# B&R Automation Studio project Installer AS Technology Solution
Automation Studio 4.9

## Logical view

### Package Logical/Libraries - Global libraries

### Program Logical/Libraries/brdkSTR

#### brdkSTR_func.h
```c
#ifndef BRDK_STR_FUNCS
#define BRDK_STR_FUNCS 1

#include <brdkSTR.h>
#include <bur/plctypes.h>

#ifdef __cplusplus
	extern "C"
	{
#endif

#ifdef __cplusplus
	};
#endif

#endif
```

#### brdkStrAToUdint.c
```c
#include <brdkSTR_func.h>

unsigned long brdkStrAToUdint(unsigned long pString, unsigned char base) {
	unsigned long value = 0;
	signed long i, len = brdkStrLen(pString);
	if(len > 0) {
		for(i=0; i <len; i++) {
			switch(base) {

				case 0: case 10:
					if(((char*)pString)[i] >= 0x30 && ((char*)pString)[i] <= 0x39) value = (value * 10) + (((char*)pString)[i]-0x30);			/* 0x30 = 0, 0x39 = 9 */
					else {
						value = 0;
						i = len;
					}
					break;

				case 2:
					if(((char*)pString)[i] >= 0x30 && ((char*)pString)[i] <= 0x31) value += (((char*)pString)[i]-0x30)*(1<<(len-1-i));			/* 0x30 = 0, 0x31 = 1 */
					else {
						value = 0;
						i = len;
					}
					break;

				case 16:
					if(((char*)pString)[i] >= 0x30 && ((char*)pString)[i] <= 0x39) 	value += (((char*)pString)[i]-0x30)*(1<<(4*(len-1-i)));		/* 0x30 = 0, 0x39 = 9 */
					else if(((char*)pString)[i] >= 0x41 && ((char*)pString)[i] <= 0x46) value += (((char*)pString)[i]-0x37)*(1<<(4*(len-1-i)));	/* 0x41 = A, 0x46 = F */
					else if(((char*)pString)[i] >= 0x61 && ((char*)pString)[i] <= 0x66)value += (((char*)pString)[i]-0x57)*(1<<(4*(len-1-i)));	/* 0x61 = a, 0x66 = f */
					else {
						value = 0;
						i = len;
					}
					break;

				default:
					value = 0;
					i = len;
					break;

			}
		}
	}
	return value;
}
```

#### brdkStrSearch.c
```c
#include <brdkSTR_func.h>

signed long brdkStrSearch(unsigned long pString, unsigned long pSearchString) {
	signed long pos=-1, i=0,j=0, len1 = brdkStrLen(pString), len2 = brdkStrLen(pSearchString);

	if(len1>len2) {
		for(i=0; i <= len1-len2; i++) {
			j=0;
			if(((char*)pString)[i] == ((char*)pSearchString)[j]) {
				while(((char*)pString)[i+j] == ((char*)pSearchString)[j]) {
					j++;
					if(j==len2) {
						pos = i;
						i=len1-len2+1;
						break;
					}
				}
			}
		}
	}
	return pos;
}
```

### Library Logical/Libraries/TrkDiag (ANSIC)
Depends on: McAcpTrak

### Program Logical/Libraries/TrkPaper

#### TrkPaperShuttleControl.c
```c
#include <bur/plctypes.h>
#include <stdint.h>
#include <AsBrStr.h>

#define TRUE 1
#define FALSE 0

#ifdef __cplusplus
	extern "C"
	{
#endif
#include "TrkPaper.h"
#ifdef __cplusplus
	};
#endif

plcbit CheckValidity(char* selectedElem){
	char buf[2];
	//Get a substring of the first 3 characters
	brdkStrSubStr((uintptr_t)&buf,(uintptr_t)selectedElem,0,3);
	//Look at the start of the selectedID, if it starts with #ID then we know a shuttle has been clicked
	if(0 == brsstrcmp((uintptr_t)&buf,(uintptr_t)&"#ID")){
		return TRUE;
	}
	else{
		return FALSE;
	}
}
USINT GetIndex(char* selectedElem){
	char buf[3];
	brdkStrSubStr((uintptr_t)&buf,(uintptr_t)selectedElem,3,brdkStrLen((uintptr_t)selectedElem) - 3);
	return (USINT)brdkStrAToUdint((uintptr_t)&buf,BRDK_STR_CONVERT_DECIMAL);
}
/* Function block for handling a shuttle control provided from the paper element's selected element ID. Must be paired with the tmCore FB */
void TrkPaperShuttleControl(struct TrkPaperShuttleControl* inst)
{
	//TODO Code disabled for the moment as major type changes are occuring. Will need to revist at a future time.

//	if(inst->Valid){
//		inst->ShInfo = inst->Internal.Fbs.ShGetInfo.ShuttleInfo;
//	}
//	switch (inst->Internal.State){
//		case trkPAPER_SH_CONTROL_OFF:
//			//******************************************************************************** Off state
//			if(inst->Enable){
//				if(inst->Handle == 0){
//					inst->Error = TRUE;
//					inst->ErrorID = trkPAPER_SH_CONTROL_ERR_INVALID_HANDLE;
//
//					inst->Internal.State = trkPAPER_SH_CONTROL_ERROR;
//				}
//				else{
//					inst->Internal.CoreInt = (TpCoreInternalTyp*)inst->Handle;
//					if(inst->Internal.CoreInt->TypeID != TpCORE_CORE_TYPE_ID){
//						inst->Error = TRUE;
//						inst->ErrorID = trkPAPER_SH_CONTROL_ERR_INVALID_HANDLE;
//
//						inst->Internal.State = trkPAPER_SH_CONTROL_ERROR;
//					}
//					else{
//						inst->Active = TRUE;
//
//						inst->Internal.State = trkPAPER_SH_CONTROL_INIT;
//					}
//				}
//			}
//			break;
//		case trkPAPER_SH_CONTROL_INIT:
//			//******************************************************************************** Init state
//			if(CheckValidity(&inst->SelectedElem)){	//Checking for the validity of the selected element format
//				inst->Internal.Idx = GetIndex(&inst->SelectedElem);	//Pulling the index from the string
//				if(inst->Internal.CoreInt->Axes[inst->Internal.Idx].Present){ //Verifying that index has a valid access in it
//					inst->ErrorID = trkPAPER_SH_CONTROL_ERR_OK;
//					inst->Valid = TRUE;
//					inst->Internal.CurrentAxis = inst->Internal.CoreInt->Axes[inst->Internal.Idx].Axis;
//
//					inst->Internal.Fbs.ShGetInfo.Axis = &inst->Internal.CurrentAxis;
//					inst->Internal.Fbs.ShGetInfo.Enable = TRUE;
//
//					inst->Internal.State = trkPAPER_SH_CONTROL_IDLE;
//				}
//				else{
//					inst->ErrorID = trkPAPER_SH_CONTROL_WARN_SH_NOT_AVAIL;
//				}
//			}
//			else{
//				inst->ErrorID = trkPAPER_SH_CONTROL_WARN_NO_ELEM_FND;
//			}
//
//			break;
//		case trkPAPER_SH_CONTROL_IDLE:
//			//******************************************************************************** Get Shuttle state
//			//Need to check for if the selected element has changed
//			inst->Internal.LastIdx = inst->Internal.Idx;
//			if(CheckValidity(&inst->SelectedElem)){
//				inst->Internal.Idx = GetIndex(&inst->SelectedElem);
//
//				if(inst->Internal.Idx != inst->Internal.LastIdx){
//					//We've changed indecies need to head back to init to reset the sh status
//					inst->Valid = FALSE;
//					inst->Internal.Fbs.ShGetInfo.Enable = FALSE;
//
//					inst->Internal.State = trkPAPER_SH_CONTROL_INIT;
//				}
//				else{
//					//Here we can start parsing commands
//					if(inst->ElasticMoveAbs){
//						//Setup the elastic move absolute block and execute it
//						inst->Internal.Fbs.ElMoveAbs.Axis = &inst->Internal.CurrentAxis;
//						inst->Internal.Fbs.ElMoveAbs.Position = inst->Parameters->Position;
//						inst->Internal.Fbs.ElMoveAbs.Velocity = inst->Parameters->Vel;
//						inst->Internal.Fbs.ElMoveAbs.Acceleration = inst->Parameters->Accel;
//						inst->Internal.Fbs.ElMoveAbs.Deceleration = inst->Parameters->Decel;
//
//						inst->Internal.Fbs.ElMoveAbs.Execute = TRUE;
//
//						inst->Internal.State = trkPAPER_SH_CONTROL_EL_MOVE_ABS;
//					}
//					else if(inst->ElasticMoveAdd){
//						//Setup the elastic move additve block and execute it
//						inst->Internal.Fbs.ElMoveAdd.Axis = &inst->Internal.CurrentAxis;
//						inst->Internal.Fbs.ElMoveAdd.Distance = inst->Parameters->Distance;
//						inst->Internal.Fbs.ElMoveAdd.Velocity = inst->Parameters->Vel;
//						inst->Internal.Fbs.ElMoveAdd.Acceleration = inst->Parameters->Accel;
//						inst->Internal.Fbs.ElMoveAdd.Deceleration = inst->Parameters->Decel;
//
//						inst->Internal.Fbs.ElMoveAdd.Execute = TRUE;
//
//						inst->Internal.State = trkPAPER_SH_CONTROL_EL_MOVE_ADD;
//					}//End of commands check conditionals
//				}
//			}
//			else{//We've received an invalid selection, need to reset the flags and Sh Status
//				inst->Valid = FALSE;
//				inst->Internal.Fbs.ShGetInfo.Enable = FALSE;
//
//				inst->Internal.State = trkPAPER_SH_CONTROL_INIT;
//			}
//
//			break;
//		case trkPAPER_SH_CONTROL_EL_MOVE_ABS:
//			//******************************************************************************** Elastic Move absolute state
//			if(inst->Internal.Fbs.ElMoveAbs.Error){
//				inst->Error = TRUE;
//				inst->ErrorID = trkPAPER_SH_CONTROL_ERR_EL_MOVE;
//
//				inst->Internal.State = trkPAPER_SH_CONTROL_ERROR;
//			}
//			else if(inst->Internal.Fbs.ElMoveAbs.Active){
//				inst->MovementActive = TRUE;
//				inst->Internal.Fbs.ElMoveAbs.Execute = FALSE;
//
//				inst->Internal.LastIdx = inst->Internal.Idx;
//				if(CheckValidity(&inst->SelectedElem)){
//					inst->Internal.Idx = GetIndex(&inst->SelectedElem);
//
//					if(inst->Internal.Idx != inst->Internal.LastIdx){
//						//We've changed indecies need to head back to init to reset the sh status
//						inst->Valid = FALSE;
//						inst->Internal.Fbs.ShGetInfo.Enable = FALSE;
//
//						inst->Internal.State = trkPAPER_SH_CONTROL_INIT;
//					}
//				}
//			}
//			else if(inst->Internal.Fbs.ElMoveAbs.Done){
//				inst->Internal.Fbs.ElMoveAbs.Execute = FALSE;
//				inst->MovementActive = FALSE;
//				inst->MovementDone = TRUE;
//
//				inst->Internal.State = trkPAPER_SH_CONTROL_MOVE_DONE;
//			}
//			break;
//		case trkPAPER_SH_CONTROL_EL_MOVE_ADD:
//			//******************************************************************************** Elastic Move Additive state
//			if(inst->Internal.Fbs.ElMoveAdd.Error){
//				inst->Error = TRUE;
//				inst->ErrorID = trkPAPER_SH_CONTROL_ERR_EL_MOVE;
//
//				inst->Internal.State = trkPAPER_SH_CONTROL_ERROR;
//			}
//			else if(inst->Internal.Fbs.ElMoveAdd.Done){
//				inst->MovementActive = FALSE;
//				inst->MovementDone = TRUE;
//
//				inst->Internal.Fbs.ElMoveAdd.Execute = FALSE;
//
//				inst->Internal.State = trkPAPER_SH_CONTROL_MOVE_DONE;
//			}
//			else{
//				inst->MovementActive = TRUE;
//			}
//			break;
//		case trkPAPER_SH_CONTROL_MOVE_DONE:
//			//******************************************************************************** Movement Done State
//			if(!inst->ElasticMoveAbs
//				&& !inst->ElasticMoveAdd){
//				inst->MovementDone = FALSE;
//
//				inst->Internal.State = trkPAPER_SH_CONTROL_IDLE;
//			}
//			break;
//		case trkPAPER_SH_CONTROL_ERROR:
//			//******************************************************************************** Error State
//			if(!inst->Enable){
//				inst->Error = FALSE;
//				inst->ErrorID = trkPAPER_SH_CONTROL_ERR_OK;
//
//				inst->Internal.Fbs.ElMoveAbs.Execute = FALSE;
//				inst->Internal.Fbs.ElMoveAdd.Execute = FALSE;
//				inst->Internal.Fbs.ShGetInfo.Enable = FALSE;
//
//				inst->Internal.Idx = 0;
//				inst->Internal.LastIdx = 0;
//
//				inst->Internal.State = trkPAPER_SH_CONTROL_OFF;
//			}
//			break;
//	}
//	//FB calls
//
//	MC_BR_ShReadInfo_AcpTrak(&inst->Internal.Fbs.ShGetInfo);
//	MC_BR_ElasticMoveAbs_AcpTrak(&inst->Internal.Fbs.ElMoveAbs);
//	MC_BR_ElasticMoveAdd_AcpTrak(&inst->Internal.Fbs.ElMoveAdd);
}
```

### Program Logical/Source/Diagnostic/TrakDiag (IEC)

#### Exit.st
```iecst
PROGRAM _EXIT
			(* Insert code here *)

END_PROGRAM
```

#### Init.st
```iecst
PROGRAM _INIT

	SegDefinition;

	paperCore.SegmentCount := TrakDiag.Seg.SegCount;
	paperCore.Segments := ADR(TrakDiag.Seg.SegList);
	paperCore.Options := ADR(paperOptions);
	paperCore.Enable := TRUE;
	paperCore.Assembly := ADR(DiagInterface.SampleTrak);
	paperCore.ShuttleMon := ADR(DiagInterface.ShuttleMon);
	paperCore.TrakStatus := ADR(TrakDiag);

	paperOptions.Color.Offset := SIZEOF(UDINT);
	paperOptions.Segment.Enabled := TRUE;
	paperOptions.Shuttle.Enabled := TRUE;
	paperOptions.Color.Enabled := TRUE;
END_PROGRAM
```

- Visualisation Logical/mappView (not shown)

Listed in the project but not available here: Logical/Libraries/TrkDiag/TrkDiag.typ, Logical/Libraries/TrkDiag/TrkDiag.var, Logical/Libraries/TrkDiag/TrkDiag.fun
